Universal Robots PolyScope program: weigh_single.urp

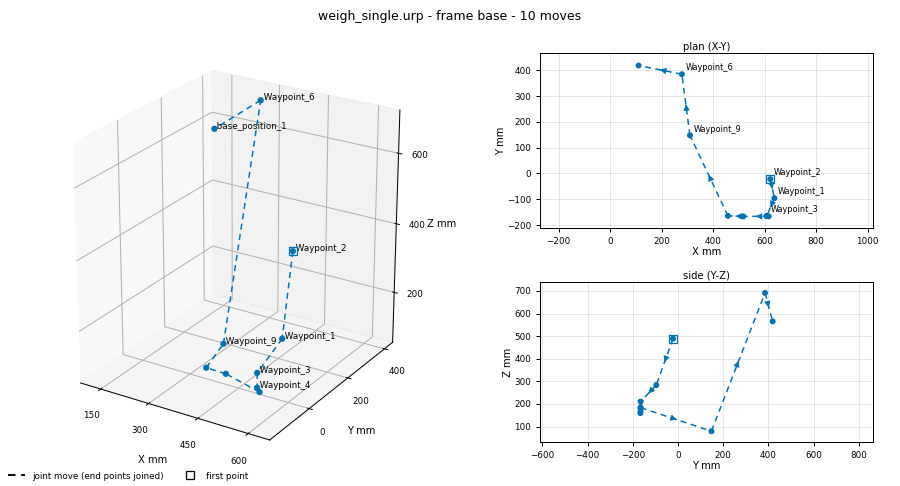
[picture p0: tool path of weigh_single.urp in frame base, 10 of 10 moves have a stored position in this frame; points joined in program order, loops and branches not executed]
Program weigh_single (installation=default directory=/programs/Nicolas_Arteaga/quality createdIn=5.12.4.1101661 lastSavedIn=5.12.4.1101661 robotSerialNumber=20225502378)
Calibrated DH parameters: a=[0.00022, -0.425328, -0.389701, 0.000059, 0.000065, 0]; d=[0.162608, 0.803456, 9.992211, -10.662202, 0.099702, 0.099559]; alpha=[1.570756, 0.001543, 0.004316, 1.570651, -1.570122, 0]; deltaTheta=[0, 0.002917, 0.116094, -0.119008, 0, -0.000001]
Robot Program (runOnlyOnce=true)
  MoveJ speed 60 deg/s, acceleration 80 deg/s^2 (useActiveTCP=true) feature=Base
    Waypoint Waypoint_2: TCP in base x=622.09 y=-21.999 z=488.949 mm, rx=0.729 ry=1.5781 rz=1.7949 rad; joints [135.515, -94.567, 106.176, -67.801, 9.2, 55.784] deg; TCP offset x=0 y=0 z=191.5 mm, rx=0 ry=0 rz=0 rad
    Waypoint Waypoint_1: TCP in base x=637.825 y=-95.931 z=283.355 mm, rx=1.2165 ry=1.151 rz=1.1657 rad; joints [145.529, -90.424, 122.897, -34.058, 59.252, 0.492] deg
    Waypoint Waypoint_3: TCP in base x=607.929 y=-165.259 z=210.32 mm, rx=1.2164 ry=1.151 rz=1.1657 rad; joints [132.864, -83.639, 129.414, -47.669, 46.63, 0.933] deg
    Waypoint Waypoint_4: TCP in base x=607.939 y=-165.205 z=168.973 mm, rx=1.2164 ry=1.1511 rz=1.1658 rad; joints [132.859, -78.034, 131.663, -55.503, 46.638, 0.907] deg
    URCap Gripper (Robotiq_Grippers, Robotiq Inc.) dataModel(position=80.0, force=100.0, speed=100.0, positionInDouble=80.0, forceInDouble=100.0, speedInDouble=100.0, slaveIds=[9], blocking=true)
    Waypoint Waypoint_7: TCP in base x=615.805 y=-166.437 z=159.387 mm, rx=1.2166 ry=1.151 rz=1.1657 rad; joints [133.72, -75.773, 130.845, -56.911, 47.515, 0.864] deg
    Wait Sleep waitTime=1
    Waypoint Waypoint_5: TCP in base x=516.967 y=-166.443 z=183.399 mm, rx=1.2166 ry=1.151 rz=1.1657 rad; joints [117.405, -91.076, 143.444, -55.007, 31.2, 1.846] deg
    Waypoint Waypoint_8: TCP in base x=457.44 y=-164.442 z=183.408 mm, rx=1.2116 ry=1.1589 rz=1.1739 rad; joints [101.707, -100.388, 151.213, -56.163, 14.906, 4.715] deg
    URCap Gripper (Robotiq_Grippers, Robotiq Inc.) dataModel(position=100.0, force=100.0, speed=100.0, positionInDouble=100.0, forceInDouble=100.0, speedInDouble=100.0, slaveIds=[9], blocking=true)
    Waypoint Waypoint_9: TCP in base x=310.148 y=147.978 z=79.403 mm, rx=-0.6951 ry=2.3951 rz=0.8204 rad; joints [132.938, -126.018, 154.738, -96.192, -47.884, 1.843] deg
    Waypoint Waypoint_6: TCP in base x=278.734 y=385.121 z=691.066 mm, rx=-0.517 ry=1.1123 rz=1.6333 rad; joints [180.614, -126.096, 113.581, -55.011, 31.191, 1.845] deg
    Waypoint base_position_1: TCP in base x=110.839 y=418.881 z=565.194 mm, rx=-1.5602 ry=-0.9892 rz=-1.3623 rad; joints [201.946, -128.864, 99.356, 35.835, 42.385, 90.241] deg
    'Finish Pressure Measurements'
